{attribute addProperty BoxType "EK1960-0000-0019"}
{attribute addProperty Id "Module_1_Channel_1_Standard_Output_X5_1AT %Q*BOOL811Module_1_Channel_2_Standard_Output_X5_2AT %Q*BOOL812Module_1_Channel_3_Standard_Output_X5_3AT %Q*BOOL813Module_1_Channel_4_Standard_Output_X5_4AT %Q*BOOL814Module_2_Channel_1_Standard_Output_X5_5AT %Q*BOOL811Module_2_Channel_2_Standard_Output_X5_6AT %Q*BOOL812Module_2_Channel_3_Standard_Output_X5_7AT %Q*BOOL813Module_2_Channel_4_Standard_Output_X5_8AT %Q*BOOL814Module_3_Channel_1_Standard_Output_X7_1AT %Q*BOOL811Module_3_Channel_2_Standard_Output_X7_2AT %Q*BOOL812Module_3_Channel_3_Standard_Output_X7_3AT %Q*BOOL813Module_3_Channel_4_Standard_Output_X7_4AT %Q*BOOL814Module_4_Channel_1_Standard_Output_X7_5AT %Q*BOOL811Module_4_Channel_2_Standard_Output_X7_6AT %Q*BOOL812Module_4_Channel_3_Standard_Output_X7_7AT %Q*BOOL813Module_4_Channel_4_Standard_Output_X7_8AT %Q*BOOL814Module_5_Channel_1_Standard_Output_X9_1AT %Q*BOOL811Module_5_Channel_2_Standard_Output_X9_2AT %Q*BOOL812Module_5_Channel_3_Standard_Output_X9_3AT %Q*BOOL813Module_5_Channel_4_Standard_Output_X9_4AT %Q*BOOL814Module_6_Channel_1_Standard_Output_X9_5AT %Q*BOOL811Module_6_Channel_2_Standard_Output_X9_6AT %Q*BOOL812Module_6_Channel_3_Standard_Output_X9_7AT %Q*BOOL813Module_6_Channel_4_Standard_Output_X9_8AT %Q*BOOL814Relais_Module_Channel_1_Standard_Output_X4_1_X4_5AT %Q*BOOL811Relais_Module_Channel_2_Standard_Output_X4_2_X4_6AT %Q*BOOL812Relais_Module_Channel_3_Standard_Output_X4_3_X4_7AT %Q*BOOL813Relais_Module_Channel_4_Standard_Output_X4_4_X4_8AT %Q*BOOL814"}
{attribute addProperty CRC "2953529769"}
{attribute addProperty SizeInBites "224"}
{attribute addProperty SizeInBytes "28"}
TYPE Outputs_B00B49A9 :
STRUCT
	{attribute addProperty Name "Module_1_Channel_1_Standard_Output_X5_1"}
	Module_1_Channel_1_Standard_Output_X5_1 AT %Q* : BOOL;
	{attribute addProperty Name "Module_1_Channel_2_Standard_Output_X5_2"}
	Module_1_Channel_2_Standard_Output_X5_2 AT %Q* : BOOL;
	{attribute addProperty Name "Module_1_Channel_3_Standard_Output_X5_3"}
	Module_1_Channel_3_Standard_Output_X5_3 AT %Q* : BOOL;
	{attribute addProperty Name "Module_1_Channel_4_Standard_Output_X5_4"}
	Module_1_Channel_4_Standard_Output_X5_4 AT %Q* : BOOL;
	{attribute addProperty Name "Module_2_Channel_1_Standard_Output_X5_5"}
	Module_2_Channel_1_Standard_Output_X5_5 AT %Q* : BOOL;
	{attribute addProperty Name "Module_2_Channel_2_Standard_Output_X5_6"}
	Module_2_Channel_2_Standard_Output_X5_6 AT %Q* : BOOL;
	{attribute addProperty Name "Module_2_Channel_3_Standard_Output_X5_7"}
	Module_2_Channel_3_Standard_Output_X5_7 AT %Q* : BOOL;
	{attribute addProperty Name "Module_2_Channel_4_Standard_Output_X5_8"}
	Module_2_Channel_4_Standard_Output_X5_8 AT %Q* : BOOL;
	{attribute addProperty Name "Module_3_Channel_1_Standard_Output_X7_1"}
	Module_3_Channel_1_Standard_Output_X7_1 AT %Q* : BOOL;
	{attribute addProperty Name "Module_3_Channel_2_Standard_Output_X7_2"}
	Module_3_Channel_2_Standard_Output_X7_2 AT %Q* : BOOL;
	{attribute addProperty Name "Module_3_Channel_3_Standard_Output_X7_3"}
	Module_3_Channel_3_Standard_Output_X7_3 AT %Q* : BOOL;
	{attribute addProperty Name "Module_3_Channel_4_Standard_Output_X7_4"}
	Module_3_Channel_4_Standard_Output_X7_4 AT %Q* : BOOL;
	{attribute addProperty Name "Module_4_Channel_1_Standard_Output_X7_5"}
	Module_4_Channel_1_Standard_Output_X7_5 AT %Q* : BOOL;
	{attribute addProperty Name "Module_4_Channel_2_Standard_Output_X7_6"}
	Module_4_Channel_2_Standard_Output_X7_6 AT %Q* : BOOL;
	{attribute addProperty Name "Module_4_Channel_3_Standard_Output_X7_7"}
	Module_4_Channel_3_Standard_Output_X7_7 AT %Q* : BOOL;
	{attribute addProperty Name "Module_4_Channel_4_Standard_Output_X7_8"}
	Module_4_Channel_4_Standard_Output_X7_8 AT %Q* : BOOL;
	{attribute addProperty Name "Module_5_Channel_1_Standard_Output_X9_1"}
	Module_5_Channel_1_Standard_Output_X9_1 AT %Q* : BOOL;
	{attribute addProperty Name "Module_5_Channel_2_Standard_Output_X9_2"}
	Module_5_Channel_2_Standard_Output_X9_2 AT %Q* : BOOL;
	{attribute addProperty Name "Module_5_Channel_3_Standard_Output_X9_3"}
	Module_5_Channel_3_Standard_Output_X9_3 AT %Q* : BOOL;
	{attribute addProperty Name "Module_5_Channel_4_Standard_Output_X9_4"}
	Module_5_Channel_4_Standard_Output_X9_4 AT %Q* : BOOL;
	{attribute addProperty Name "Module_6_Channel_1_Standard_Output_X9_5"}
	Module_6_Channel_1_Standard_Output_X9_5 AT %Q* : BOOL;
	{attribute addProperty Name "Module_6_Channel_2_Standard_Output_X9_6"}
	Module_6_Channel_2_Standard_Output_X9_6 AT %Q* : BOOL;
	{attribute addProperty Name "Module_6_Channel_3_Standard_Output_X9_7"}
	Module_6_Channel_3_Standard_Output_X9_7 AT %Q* : BOOL;
	{attribute addProperty Name "Module_6_Channel_4_Standard_Output_X9_8"}
	Module_6_Channel_4_Standard_Output_X9_8 AT %Q* : BOOL;
	{attribute addProperty Name "Relais_Module_Channel_1_Standard_Output_X4_1_X4_5"}
	Relais_Module_Channel_1_Standard_Output_X4_1_X4_5 AT %Q* : BOOL;
	{attribute addProperty Name "Relais_Module_Channel_2_Standard_Output_X4_2_X4_6"}
	Relais_Module_Channel_2_Standard_Output_X4_2_X4_6 AT %Q* : BOOL;
	{attribute addProperty Name "Relais_Module_Channel_3_Standard_Output_X4_3_X4_7"}
	Relais_Module_Channel_3_Standard_Output_X4_3_X4_7 AT %Q* : BOOL;
	{attribute addProperty Name "Relais_Module_Channel_4_Standard_Output_X4_4_X4_8"}
	Relais_Module_Channel_4_Standard_Output_X4_4_X4_8 AT %Q* : BOOL;
END_STRUCT
END_TYPE

(* stored: Version 1.2.0.0, ProductVersion 3.1.4024.9
   DUT Outputs_B00B49A9: Id {8d31ae49-c030-40a3-8a97-5ed8d8d1d985} *)
